SUBAPPLICATION PlusPlus (* Subapplication Type *)
  (* Standard: 61499-2 *)
  (* Version 1.0, 2023-02-17, Franz *)
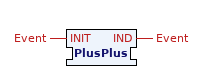
  EVENT_INPUT
    INIT;
  END_EVENT
  EVENT_OUTPUT
    IND;
  END_EVENT
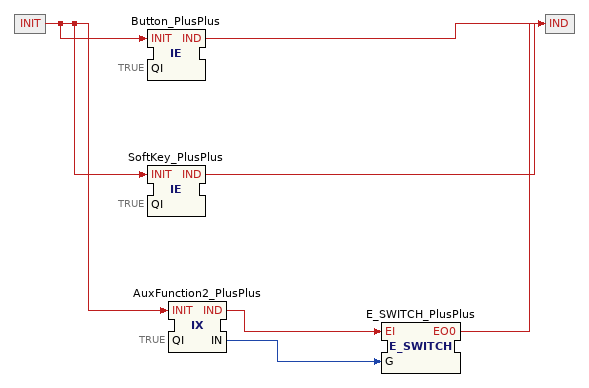
  FBS
    Button_PlusPlus : IE(QI := TRUE);
    SoftKey_PlusPlus : IE(QI := TRUE);
    AuxFunction2_PlusPlus : IX(QI := TRUE);
    E_SWITCH_PlusPlus : E_SWITCH;
  END_FBS
  EVENT_CONNECTIONS
    INIT TO Button_PlusPlus.INIT;
    Button_PlusPlus.IND TO IND;
    INIT TO SoftKey_PlusPlus.INIT;
    SoftKey_PlusPlus.IND TO IND;
    INIT TO AuxFunction2_PlusPlus.INIT;
    AuxFunction2_PlusPlus.IND TO E_SWITCH_PlusPlus.EI;
    E_SWITCH_PlusPlus.EO0 TO IND;
  END_CONNECTIONS
  DATA_CONNECTIONS
    AuxFunction2_PlusPlus.IN TO E_SWITCH_PlusPlus.G;
  END_CONNECTIONS
END_SUBAPPLICATION
